{attribute 'strict'}
{attribute 'to_string'}
TYPE E_MessageType :
(
  eMessageEmpty,
  eMessageVerbose,
  eMessageInfo,
  eMessageWarn,
  eMessageError
)DINT;
END_TYPE

(* stored: Version 1.1.0.1, ProductVersion 3.1.4024.12
   DUT E_MessageType: Id {7f8d3eda-1f44-4db9-b42c-d0e3626f5bdc} *)
